(* IEC 61131-3 sources: volt/packages/volt-lsp-iec/test-corpus/bakon-nano/Device/Plc Logic/Application/Library Manager/(unresolved)/datasources interfaces, 60 files *)

(* ---- BYTEORDER.dut ---- *)
TYPE BYTEORDER :
(
	UNKNOWN,
	HOST,
	INTEL,
	MOTOROLA
);
END_TYPE

(* ---- ETRACEADDRESSFLAGS.dut ---- *)
TYPE ETRACEADDRESSFLAGS :
(
	IEC := 16#1,
	IOCONFIG := 16#2,
	AREAOFFSET := 16#20,
	PROP := 16#40
);
END_TYPE

(* ---- ITEMACCESS.dut ---- *)
TYPE ITEMACCESS :
(
	NONE,
	READ,
	READWRITE
);
END_TYPE

(* ---- ITEMNAME.dut ---- *)
TYPE ITEMNAME :
STRUCT
	NAMETYPE : ItemNameType;
	NAMEDATA : POINTER TO BYTE;
END_STRUCT
END_TYPE

(* ---- ITEMNAMETYPE.dut ---- *)
TYPE ITEMNAMETYPE :
(
	NORMALSTRING
);
END_TYPE

(* ---- ITEMQUALITY.dut ---- *)
TYPE ITEMQUALITY :
(
	NEW,
	GOOD,
	BAD
);
END_TYPE

(* ---- MONITORINGSTATE.dut ---- *)
TYPE MONITORINGSTATE :
(
	INITIALIZED,
	CONNECTING,
	CONNECTED,
	SHUTTINGDOWN,
	SHUTDOWN,
	WAITINGFORRECONNECT,
	WAITINGFORCOMMSETTING,
	UNKNOWN
);
END_TYPE

(* ---- PERSISTANTITEMLISTUSAGE.dut ---- *)
TYPE PERSISTANTITEMLISTUSAGE :
(
	UNSPECIFIED,
	RECIPES
);
END_TYPE

(* ---- REPLACEMENTINFO.dut ---- *)
TYPE REPLACEMENTINFO :
STRUCT
	PPARENTREPLACEMENTINFO : POINTER TO ReplacementInfo;
	ARRNAME : POINTER TO ARRAY [0..0] OF POINTER TO STRING(255);
	ARRREPLACEMENT : POINTER TO ARRAY [0..0] OF POINTER TO STRING(255);
	NCOUNT : INT;
END_STRUCT
END_TYPE

(* ---- REUSABLEREQUESTOPERATIONS.dut ---- *)
TYPE REUSABLEREQUESTOPERATIONS :
(
	PREPARE,
	READ,
	WRITE
);
END_TYPE

(* ---- ERRORS.gvl ---- *)
VAR_GLOBAL
	ERR_DS_UNKNOWN : UDINT := 16#2000;
	ERR_DS_UNKNOWN_GROUP : UDINT := 16#2001;
	ERR_DS_UNKNOWN_SYMBOL : UDINT := 16#2002;
	ERR_DS_UNKNOWN_TRANSACTION : UDINT := 16#2003;
	ERR_DS_INVALID_STATE : UDINT := 16#2004;
	ERR_DS_INVALID_PATH : UDINT := 16#2005;
	ERR_DS_SOURCENOTFOUND : UDINT := 16#2006;
	ERR_DS_ITEMNOTFOUND : UDINT := 16#2007;
	ERR_DS_MULTITASKING_LOCKED : UDINT := 16#2008;
	ERR_DS_TIMEOUT : UDINT := 16#2009;
	ERR_DS_BADITEMS : UDINT := 16#200A;
	ERR_DS_ITEMNOTACTIVE : UDINT := 16#200B;
	ERR_DS_RETRYLOGIN : UDINT := 16#200C;
	ERR_DS_READONLY_ITEM : UDINT := 16#200D;
	ERR_DS_DATASOURCE_INDEX_MISMATCH : UDINT := 16#200E;
	ERR_DSD_IDENTITY_MISMATCH : UDINT := 16#2100;
	ERR_DSD_LOGINFAILED : UDINT := 16#2101;
	ERR_DSD_LOGINNECESSARY : UDINT := 16#2102;
	ERR_DSD_BUSY : UDINT := 16#2103;
	ERR_DSD_NOTREACHABLE : UDINT := 16#2104;
	ERR_DSD_DUPLICATE : UDINT := 16#2105;
	ERR_DSD_NOSYMBOLS : UDINT := 16#2106;
	ERR_DSD_CONNECTIONLOST : UDINT := 16#2107;
	ERR_DSD_CONNECTIONDENIED : UDINT := 16#2108;
	ERR_DSD_CONNECTIONDENIED_SRVRESOURCES : UDINT := 16#2109;
	ERR_DSD_PROTOCOL_MISMATCH : UDINT := 16#210A;
	ERR_DSD_LOGIN_NOTPOSSIBLE : UDINT := 16#210B;
	ERR_DSI_FAILED : UDINT := 16#2200;
	ERR_DSI_MISSING_GETACCESSOR : UDINT := 16#2201;
	ERR_DSI_MISSING_SETACCESSOR : UDINT := 16#2202;
	ERR_DSI_UNEXPECTED_ADDRESSINFO : UDINT := 16#2203;
	ERR_DSI_COMMBUFFEROVERRUN : UDINT := 16#2204;
	ERR_DSI_TOOMANYITEMS : UDINT := 16#2205;
	ERR_DSI_DATAMISSING : UDINT := 16#2206;
	ERR_DSI_ITEMNOTFOUND : UDINT := 16#2207;
	ERR_DSI_CONNECTIONLOST : UDINT := 16#2208;
	ERR_DSI_PROTOCOLSPECIFIC_ERROR_RANGESTART : UDINT := 16#2300;
	ERR_DSI_PROTOCOLSPECIFIC_ERROR_RANGEEND : UDINT := 16#23FF;
END_VAR

(* ---- ICDSV3REQUEST.itf ---- *)
INTERFACE ICDSV3REQUEST
END_INTERFACE

METHOD SETCONTENTDATA : SysTypes.RTS_IEC_RESULT
VAR_INPUT
	PDATA : POINTER TO BYTE;
	UXISIZE : __UXINT;
END_VAR
END_METHOD

(* ---- ICDSV3REQUESTHANDLING.itf ---- *)
INTERFACE ICDSV3REQUESTHANDLING
END_INTERFACE

METHOD CREATECDSV3REQUEST : ICDSV3Request
VAR_INPUT
	UISERVICEGROUP : UINT;
	UISERVICE : UINT;
END_VAR
END_METHOD

(* ---- ICDSV3RESPONSE.itf ---- *)
INTERFACE ICDSV3RESPONSE
END_INTERFACE

(* ---- ICDSV3SERVICEWRITER.itf ---- *)
INTERFACE ICDSV3SERVICEWRITER
END_INTERFACE

(* ---- ICREDENTIALS.itf ---- *)
INTERFACE ICREDENTIALS
END_INTERFACE

(* ---- ICREDENTIALSPROVIDER.itf ---- *)
INTERFACE ICREDENTIALSPROVIDER
END_INTERFACE

METHOD GETCREDENTIALS : SysTypes.RTS_IEC_RESULT
VAR_INPUT
	UXIREQUESTID : __UXINT;
END_VAR
VAR_OUTPUT
	CREDENTIALS : ICredentials;
END_VAR
END_METHOD

METHOD ISGETCREDENTIALSFINISHED : SysTypes.RTS_IEC_RESULT
VAR_INPUT
	UXIREQUESTID : __UXINT;
END_VAR
END_METHOD

METHOD LOGINFAILED : SysTypes.RTS_IEC_RESULT
VAR_INPUT
	UXIREQUESTID : __UXINT;
END_VAR
VAR_OUTPUT
	TRETRYWAITTIME : TIME;
END_VAR
END_METHOD

METHOD LOGINSUCCEEDED
VAR_INPUT
	UXIREQUESTID : __UXINT;
END_VAR
END_METHOD

METHOD STARTGETCREDENTIALS : __UXINT
VAR_INPUT
	PSTDATASOURCE : POINTER TO STRING;
END_VAR
VAR_OUTPUT
	UDIERRORCODE : SysTypes.RTS_IEC_RESULT;
END_VAR
END_METHOD

(* ---- ICREDENTIALSUSERPASSWORD.itf ---- *)
INTERFACE ICREDENTIALSUSERPASSWORD
END_INTERFACE

(* ---- ICUSTOMREQUEST.itf ---- *)
INTERFACE ICUSTOMREQUEST
END_INTERFACE

(* ---- ICUSTOMREQUESTCALLBACK.itf ---- *)
INTERFACE ICUSTOMREQUESTCALLBACK
END_INTERFACE

METHOD REQUESTFINISHED
VAR_INPUT
	REQUEST : ICustomRequest;
	RESPONSE : ICustomResponse;
	RESULT : SysTypes.RTS_IEC_RESULT;
END_VAR
END_METHOD

(* ---- ICUSTOMREQUESTHANDLING.itf ---- *)
INTERFACE ICUSTOMREQUESTHANDLING
END_INTERFACE

METHOD RELEASEREQUEST : SysTypes.RTS_IEC_RESULT
VAR_INPUT
	REQUEST : ICustomRequest;
END_VAR
END_METHOD

(* ---- ICUSTOMRESPONSE.itf ---- *)
INTERFACE ICUSTOMRESPONSE
END_INTERFACE

(* ---- IDATAITEM.itf ---- *)
INTERFACE IDATAITEM
END_INTERFACE

METHOD SETERROR
VAR_INPUT
	ERRORCODE : SysTypes.RTS_IEC_RESULT;
END_VAR
END_METHOD

(* ---- IDATAITEMBASE.itf ---- *)
INTERFACE IDATAITEMBASE
END_INTERFACE

(* ---- IDATAITEMLIST.itf ---- *)
INTERFACE IDATAITEMLIST
END_INTERFACE

METHOD CLEAR : SysTypes.RTS_IEC_RESULT
END_METHOD

METHOD CREATEANDADD : SysTypes.RTS_IEC_RESULT
VAR_INPUT
	PSTSYMBOL : POINTER TO STRING;
END_VAR
END_METHOD

METHOD GETITEM : IDataItemBase
VAR_INPUT
	UDIINDEX : UDINT;
END_VAR
END_METHOD

(* ---- IDATAITEMLISTEXPANDING.itf ---- *)
INTERFACE IDATAITEMLISTEXPANDING
END_INTERFACE

METHOD CREATEANDADDEXPANDING : SysTypes.RTS_IEC_RESULT
VAR_INPUT
	PSTSYMBOL : POINTER TO STRING;
END_VAR
END_METHOD

(* ---- IDATAITEMLISTPERSISTANT.itf ---- *)
INTERFACE IDATAITEMLISTPERSISTANT
END_INTERFACE

METHOD FINISHEDADDING : SysTypes.RTS_IEC_RESULT
END_METHOD

(* ---- IDATAITEMVALUEASSIGNER.itf ---- *)
INTERFACE IDATAITEMVALUEASSIGNER
END_INTERFACE

METHOD GETRAWVALUE : POINTER TO BYTE
END_METHOD

METHOD SETRAWVALUE
VAR_INPUT
	PDATA : POINTER TO BYTE;
END_VAR
END_METHOD

(* ---- IDATASOURCE.itf ---- *)
INTERFACE IDATASOURCE
END_INTERFACE

METHOD ENQUEUECUSTOMREQUEST : SysTypes.RTS_IEC_RESULT
VAR_INPUT
	REQUEST : ICustomRequest;
	FINISHEDCALLBACK : ICustomRequestCallback;
END_VAR
END_METHOD

METHOD SETCREDENTIALSPROVIDER : SysTypes.RTS_IEC_RESULT
VAR_INPUT
	PROVIDER : ICredentialsProvider;
END_VAR
END_METHOD

(* ---- IDATASOURCE2.itf ---- *)
INTERFACE IDATASOURCE2
END_INTERFACE

(* ---- IDATASOURCE3.itf ---- *)
INTERFACE IDATASOURCE3
END_INTERFACE

METHOD SETUPDATERATEREDUCTION
VAR_INPUT
	UIFACTOR : UINT;
	TMAXVALUE : TIME;
END_VAR
END_METHOD

(* ---- IDATASOURCESACTIONRECORD.itf ---- *)
INTERFACE IDATASOURCESACTIONRECORD
END_INTERFACE

(* ---- IDATASOURCESFRAMEMANAGER.itf ---- *)
INTERFACE IDATASOURCESFRAMEMANAGER
END_INTERFACE

METHOD GETCOUNT : INT
END_METHOD

METHOD GETREPLACEDPATH : POINTER TO STRING(255)
VAR_INPUT
	PSTINTERFACEVAR : POINTER TO STRING(255);
	PREPLACEMENTINFO : POINTER TO ReplacementInfo;
END_VAR
END_METHOD

METHOD GETREPLACEMENTINFO : POINTER TO ReplacementInfo
VAR_INPUT
	PSTFRAMEPATH : POINTER TO STRING(255);
END_VAR
END_METHOD

(* ---- IDATASOURCESMGR.itf ---- *)
INTERFACE IDATASOURCESMGR
END_INTERFACE

METHOD ACTIONRECORDDELETE : SysTypes.RTS_IEC_RESULT
VAR_INPUT
	RECORD : IDatasourcesActionRecord;
END_VAR
END_METHOD

METHOD ACTIONRECORDREPLAY : SysTypes.RTS_IEC_RESULT
VAR_INPUT
	RECORD : IDatasourcesActionRecord;
END_VAR
END_METHOD

METHOD ACTIONRECORDINGGETRESULT : SysTypes.RTS_IEC_RESULT
VAR_OUTPUT
	RESULT : IDatasourcesActionRecord;
END_VAR
END_METHOD

METHOD ACTIONRECORDINGSTART : SysTypes.RTS_IEC_RESULT
END_METHOD

METHOD ALLITEMSOK : SysTypes.RTS_IEC_RESULT
END_METHOD

METHOD BEGINDATACONFIGURATION : SysTypes.RTS_IEC_RESULT
VAR_INPUT
	XBLOCKING : BOOL;
END_VAR
END_METHOD

METHOD CREATEITEMLIST : IDataItemList
VAR_INPUT
	UDIINITIALCAPACITY : UDINT;
END_VAR
END_METHOD

METHOD DELETEITEMLIST : SysTypes.RTS_IEC_RESULT
VAR_INPUT
	ITEMSLIST : IDataItemList;
END_VAR
END_METHOD

METHOD ENDDATACONFIGURATION : SysTypes.RTS_IEC_RESULT
END_METHOD

METHOD GETDATASOURCE : IDatasource
VAR_INPUT
	NAME : STRING;
END_VAR
END_METHOD

METHOD GETITEMINFO : IDataItemBase
VAR_INPUT
	PSTSYMBOL : POINTER TO STRING;
END_VAR
END_METHOD

METHOD READITEMSSYNC : SysTypes.RTS_IEC_RESULT
VAR_INPUT
	ITEMS : IDataItemList;
END_VAR
END_METHOD

METHOD RELEASEDATA : SysTypes.RTS_IEC_RESULT
VAR_INPUT
	PSTSYMBOL : POINTER TO STRING;
END_VAR
END_METHOD

METHOD SETCREDENTIALSPROVIDER : SysTypes.RTS_IEC_RESULT
VAR_INPUT
	PROVIDER : ICredentialsProvider;
END_VAR
END_METHOD

METHOD USEDATA : SysTypes.RTS_IEC_RESULT
VAR_INPUT
	PSTSYMBOL : POINTER TO STRING;
END_VAR
END_METHOD

METHOD WRITEITEMSSYNC : SysTypes.RTS_IEC_RESULT
VAR_INPUT
	ITEMS : IDataItemList;
END_VAR
END_METHOD

(* ---- IDATASOURCESMGR2.itf ---- *)
INTERFACE IDATASOURCESMGR2
END_INTERFACE

METHOD ADDNOTIFICATIONCLIENT : SysTypes.RTS_IEC_RESULT
VAR_INPUT
	CLIENT : INotificationClient;
END_VAR
END_METHOD

METHOD CREATEPERSISTANTITEMLIST : IDataItemListPersistant
VAR_INPUT
	USAGE : PersistantItemListUsage;
	USAGEDETAILS : WSTRING;
	UDIINITIALCAPACITY : UDINT;
END_VAR
VAR_OUTPUT
	RESULT : SysTypes.RTS_IEC_RESULT;
END_VAR
END_METHOD

METHOD DELETEPERSISTANTITEMLIST
VAR_INPUT
	ITEMSLIST : IDataItemListPersistant;
END_VAR
END_METHOD

METHOD GETPERSISTANTITEMLIST : IDataItemListPersistant
VAR_INPUT
	LISTNR : INT;
END_VAR
END_METHOD

METHOD LOCK : SysTypes.RTS_IEC_RESULT
VAR_INPUT
	XBLOCKING : BOOL;
END_VAR
END_METHOD

METHOD REMOVENOTIFICATIONCLIENT : SysTypes.RTS_IEC_RESULT
VAR_INPUT
	CLIENT : INotificationClient;
END_VAR
END_METHOD

METHOD UNLOCK : SysTypes.RTS_IEC_RESULT
END_METHOD

(* ---- IDATASOURCESMGR3.itf ---- *)
INTERFACE IDATASOURCESMGR3
END_INTERFACE

METHOD USEDATAEXPANDING : SysTypes.RTS_IEC_RESULT
VAR_INPUT
	PSTSYMBOL : POINTER TO STRING;
END_VAR
END_METHOD

(* ---- IDATASOURCESMGR4.itf ---- *)
INTERFACE IDATASOURCESMGR4
END_INTERFACE

METHOD GETDATASOURCEITFBYINDEX : IDatasource3
VAR_INPUT
	INDEX : INT;
END_VAR
END_METHOD

(* ---- IDATASOURCETRACEADDRESSINFOPROVIDER.itf ---- *)
INTERFACE IDATASOURCETRACEADDRESSINFOPROVIDER
END_INTERFACE

METHOD CREATETRACEADDRESSINFOWRITER : ITraceAddressInfoWriter
VAR_INPUT
	PSSYMBOL : POINTER TO STRING;
END_VAR
VAR_OUTPUT
	UDIRESULT : UDINT;
END_VAR
END_METHOD

METHOD GETPOINTERSIZEINBYTES : BYTE
VAR_OUTPUT
	UDIRESULT : UDINT;
END_VAR
END_METHOD

METHOD RELEASETRACEADDRESSINFOWRITER : SysTypes.RTS_IEC_RESULT
VAR_INPUT
	ITFTRACEADDRESSINFOWRITER : ITraceAddressInfoWriter;
END_VAR
END_METHOD

(* ---- IDRIVER.itf ---- *)
INTERFACE IDRIVER
END_INTERFACE

METHOD INIT
VAR_INPUT
	PCFGDATA : POINTER TO BYTE;
END_VAR
END_METHOD

(* ---- IDRIVERCDSV3.itf ---- *)
INTERFACE IDRIVERCDSV3
END_INTERFACE

METHOD CANSENDCDSV3CUSTOMREQUEST : BOOL
END_METHOD

(* ---- IDRIVERCREDENTIALSHANDLING.itf ---- *)
INTERFACE IDRIVERCREDENTIALSHANDLING
END_INTERFACE

METHOD SETCREDENTIALS : SysTypes.RTS_IEC_RESULT
VAR_INPUT
	CREDENTIALS : ICredentials;
END_VAR
END_METHOD

(* ---- IDRIVERCREDENTIALSHANDLINGEVERYLOGIN.itf ---- *)
INTERFACE IDRIVERCREDENTIALSHANDLINGEVERYLOGIN
END_INTERFACE

(* ---- IDRIVERCUSTOMREQUEST.itf ---- *)
INTERFACE IDRIVERCUSTOMREQUEST
END_INTERFACE

(* ---- IDRIVERLARGEREQUEST.itf ---- *)
INTERFACE IDRIVERLARGEREQUEST
END_INTERFACE

(* ---- IDRIVERREQUEST.itf ---- *)
INTERFACE IDRIVERREQUEST
END_INTERFACE

(* ---- IDRIVERREQUESTFACTORY.itf ---- *)
INTERFACE IDRIVERREQUESTFACTORY
END_INTERFACE

METHOD CREATEREADREQUEST : IDriverRequest
VAR_INPUT
	PITEMS : POINTER TO IDataItem;
	ITEMSCOUNT : DINT;
END_VAR
END_METHOD

METHOD CREATEWRITEREQUEST : IDriverRequest
VAR_INPUT
	PITEMS : POINTER TO IDataItem;
	ITEMSCOUNT : DINT;
END_VAR
END_METHOD

METHOD RELEASEREQUEST
VAR_INPUT
	REQUEST : IDriverRequest;
END_VAR
END_METHOD

(* ---- IDRIVERREQUESTFACTORYCUSTOM.itf ---- *)
INTERFACE IDRIVERREQUESTFACTORYCUSTOM
END_INTERFACE

METHOD CREATECUSTOMREQUEST : IDriverCustomRequest
VAR_INPUT
	REQUEST : ICustomRequest;
END_VAR
END_METHOD

(* ---- IDRIVERREQUESTFACTORYLARGEREQUESTS.itf ---- *)
INTERFACE IDRIVERREQUESTFACTORYLARGEREQUESTS
END_INTERFACE

METHOD CREATELARGEREADREQUEST : IDriverLargeRequest
VAR_INPUT
	PITEMS : POINTER TO IDataItem;
	ITEMSCOUNT : DINT;
END_VAR
END_METHOD

METHOD CREATELARGEWRITEREQUEST : IDriverLargeRequest
VAR_INPUT
	PITEMS : POINTER TO IDataItem;
	ITEMSCOUNT : DINT;
END_VAR
END_METHOD

(* ---- IDRIVERREQUESTFACTORYREUSABLE.itf ---- *)
INTERFACE IDRIVERREQUESTFACTORYREUSABLE
END_INTERFACE

METHOD CREATEREUSABLEREQUEST : IDriverRequestReusable
VAR_INPUT
	PITEMS : POINTER TO IDataItem;
	ITEMSCOUNT : DINT;
END_VAR
END_METHOD

(* ---- IDRIVERREQUESTREUSABLE.itf ---- *)
INTERFACE IDRIVERREQUESTREUSABLE
END_INTERFACE

(* ---- IDRIVERSPECIFICDATA.itf ---- *)
INTERFACE IDRIVERSPECIFICDATA
END_INTERFACE

METHOD RELEASE
END_METHOD

(* ---- IDRIVERSPECIFIEDSETTINGS.itf ---- *)
INTERFACE IDRIVERSPECIFIEDSETTINGS
END_INTERFACE

METHOD RECONNECTWAITTIME : TIME
VAR_OUTPUT
	XUSEDEFAULT : BOOL;
END_VAR
END_METHOD

METHOD TIMEOUTSYNCSHUTDOWN : TIME
VAR_OUTPUT
	XUSEDEFAULT : BOOL;
END_VAR
END_METHOD

(* ---- IDRIVERSPECIFIEDSETTINGSREADONCHANGE.itf ---- *)
INTERFACE IDRIVERSPECIFIEDSETTINGSREADONCHANGE
END_INTERFACE

(* ---- IDRIVERSTATEMACHINE.itf ---- *)
INTERFACE IDRIVERSTATEMACHINE
END_INTERFACE

METHOD CONNECTING : SysTypes.RTS_IEC_RESULT
END_METHOD

METHOD POLLREQUESTRESULT : SysTypes.RTS_IEC_RESULT
VAR_INPUT
	REQUEST : IDriverRequest;
END_VAR
END_METHOD

METHOD RESETAFTERERROR
END_METHOD

METHOD SENDREQUEST : SysTypes.RTS_IEC_RESULT
VAR_INPUT
	REQUEST : IDriverRequest;
END_VAR
END_METHOD

METHOD SHUTTINGDOWN : SysTypes.RTS_IEC_RESULT
END_METHOD

METHOD STARTCONNECT : SysTypes.RTS_IEC_RESULT
END_METHOD

METHOD STARTSHUTDOWN : SysTypes.RTS_IEC_RESULT
END_METHOD

(* ---- IDRIVERSTATEMACHINE2.itf ---- *)
INTERFACE IDRIVERSTATEMACHINE2
END_INTERFACE

METHOD WAITINGFORCOMMSETTING : SysTypes.RTS_IEC_RESULT
VAR_INPUT
	XPREVIEW : BOOL;
END_VAR
END_METHOD

(* ---- IDRIVERSTATEMACHINENOTIFYBEFORESHUTDOWN.itf ---- *)
INTERFACE IDRIVERSTATEMACHINENOTIFYBEFORESHUTDOWN
END_INTERFACE

METHOD BEFORESHUTDOWN
VAR_INPUT
	XDURINGEXIT : BOOL;
END_VAR
END_METHOD

(* ---- IDRIVERSTATEMACHINESHUTDOWNTIMEOUT.itf ---- *)
INTERFACE IDRIVERSTATEMACHINESHUTDOWNTIMEOUT
END_INTERFACE

METHOD SHUTDOWNTIMEDOUT
END_METHOD

(* ---- IDRIVERTRACEADDRESSINFOPROVIDER.itf ---- *)
INTERFACE IDRIVERTRACEADDRESSINFOPROVIDER
END_INTERFACE

METHOD CREATETRACEADDRESSINFOWRITER : ITraceAddressInfoWriter
VAR_INPUT
	ITFDATAITEM : IDataItem;
END_VAR
VAR_OUTPUT
	UDIRESULT : UDINT;
END_VAR
END_METHOD

METHOD GETPOINTERSIZEINBYTES : BYTE
END_METHOD

METHOD RELEASETRACEADDRESSINFOWRITER : SysTypes.RTS_IEC_RESULT
VAR_INPUT
	ITFTRACEADDRESSINFOWRITER : ITraceAddressInfoWriter;
END_VAR
END_METHOD

(* ---- INOTIFICATIONCLIENT.itf ---- *)
INTERFACE INOTIFICATIONCLIENT
END_INTERFACE

METHOD LISTOPERATIONDONE
VAR_INPUT
	XWRITING : BOOL;
	DATASOURCENAME : ItemName;
	RESULT : SysTypes.RTS_IEC_RESULT;
END_VAR
END_METHOD

METHOD LISTOPERATIONSTART
VAR_INPUT
	XWRITING : BOOL;
	DATASOURCENAME : ItemName;
END_VAR
END_METHOD

METHOD LISTVALUEREAD
VAR_INPUT
	REMOTENAME : ItemName;
	PREADVALUE : POINTER TO BYTE;
	VALUETYPE : IBaseLibrary.TypeClass;
	VALUESIZE : __UXINT;
END_VAR
END_METHOD

METHOD LISTVALUEWRITE
VAR_INPUT
	REMOTENAME : ItemName;
	PWRITEVALUE : POINTER TO BYTE;
	VALUETYPE : IBaseLibrary.TypeClass;
	VALUESIZE : __UXINT;
END_VAR
END_METHOD

METHOD READREQUESTDONE
VAR_INPUT
	DATASOURCENAME : ItemName;
	RESULT : SysTypes.RTS_IEC_RESULT;
END_VAR
END_METHOD

METHOD READREQUESTSTART
VAR_INPUT
	DATASOURCENAME : ItemName;
END_VAR
END_METHOD

METHOD SINGLEVALUEREAD
VAR_INPUT
	REMOTENAME : ItemName;
	PREADVALUE : POINTER TO BYTE;
	VALUETYPE : IBaseLibrary.TypeClass;
	VALUESIZE : __UXINT;
END_VAR
END_METHOD

METHOD SINGLEVALUEWRITE
VAR_INPUT
	REMOTENAME : ItemName;
	POLDVALUE : POINTER TO BYTE;
	PNEWVALUE : POINTER TO BYTE;
	VALUETYPE : IBaseLibrary.TypeClass;
	VALUESIZE : __UXINT;
END_VAR
END_METHOD

METHOD WRITEREQUESTDONE
VAR_INPUT
	DATASOURCENAME : ItemName;
	RESULT : SysTypes.RTS_IEC_RESULT;
END_VAR
END_METHOD

METHOD WRITEREQUESTSTART
VAR_INPUT
	DATASOURCENAME : ItemName;
END_VAR
END_METHOD

(* ---- ITRACEADDRESSINFOWRITER.itf ---- *)
INTERFACE ITRACEADDRESSINFOWRITER
END_INTERFACE

METHOD GETADDRESSFLAGS : ETraceAddressFlags
END_METHOD

METHOD GETSIZE : __UXINT
END_METHOD

METHOD GETTYPE : IBaseLibrary.TypeClass
END_METHOD

METHOD RELEASE
END_METHOD

METHOD WRITEADDRESSINFO : UDINT
VAR_INPUT
	ITFCDSV3SERVICEWRITER : ICDSV3ServiceWriter;
	XHASTOSWAP : BOOL;
END_VAR
END_METHOD
